{attribute 'TcGenerated'}
{attribute 'no-analysis'}
{attribute 'linkalways'}
// This function has been automatically generated from the project information.
VAR_GLOBAL CONSTANT
	{attribute 'const_non_replaced'}
	stLibVersion_Device_Library : ST_LibVersion := (iMajor := 1, iMinor := 3, iBuild := 0, iRevision := 3, nFlags := 0, sVersion := '1.3.0.3');
END_VAR

(* stored: Version 1.1.0.1, ProductVersion 3.1.4024.5
   GVL Global_Version: Id {03aef1f3-0792-0632-0249-7c58b76eda69} *)
